Fanuc KAREL source: kt00001.KL

-- PROVISIONAL review KL for V940-1; original PC SHA256 0334f2e69ae033c317190983798f348f00a7f2da37344383dd7ed481bdc51d4e
-- Incomplete behavior may be omitted. Consult companion uncertainty JSON. Do not deploy.
PROGRAM KT00001
%NOLOCKGROUP
VAR
  I1 : INTEGER
  I2 : INTEGER
  OUT : INTEGER
BEGIN
  -- V9_ZERO_TABLE_METADATA_HINT layout=0001; no indexed target words; source/name/runtime held
  -- UNRESOLVED_PC offsets 5-16; opcodes 2E,23
  -- UNRESOLVED_PC offsets 21-32; opcodes 2E,23
  -- UNRESOLVED_PC offsets 37-48; opcodes 2E,23
  -- UNRESOLVED_PC offsets 53-64; opcodes 2E,23
  -- UNRESOLVED_PC offsets 69-88; opcodes 21,21,52,23
  -- UNRESOLVED_PC offsets 93-97; opcodes 7F
END KT00001
